FUNCTION_BLOCK FB_Component_Preplate_Rack EXTENDS FB_ComponentBase_SR
VAR_INPUT
    Executing : BOOL;

END_VAR

VAR
    // Inputs

    Button  : FB_Component_Button;
    Closed  : FB_DigitalSensor;
    _InAuto : BOOL;

    // Outputs
    Lock : FB_Component_Indicator;
END_VAR

VAR
    State    : E_RackState;
    R_Button : R_TRIG;

    //Properties
    _Available   : BOOL;
    _LinkBlocked : BOOL;
    _Blocked     : BOOL;
    Linked       : BOOL := TRUE;

    // Alarms
    RackDoorAlarms : ARRAY[1..RACK_DOOR_ALARMS_COUNT] OF FB_TcAlarm;

END_VAR

VAR
    // Internal state variables
    DoorLocked : BOOL := FALSE;
END_VAR

VAR CONSTANT
    RACK_DOOR_ALARMS_COUNT : UDINT := 5;
END_VAR

METHOD Block
VAR_INPUT
    Blocked : BOOL;
END_VAR
_Blocked := Blocked;
END_METHOD

PROPERTY Blocked : BOOL
GET
Blocked := _Blocked;
END_GET
SET
_Blocked := Blocked;
END_SET
END_PROPERTY

//! @summary This method serves as the entry point for all underlying FB logic
METHOD PUBLIC CyclicLogic

//! @description This method should be called cyclically by descendant function blocks by invoking <c>SUPER^.CyclicLogic()</c>.  Alternatively, the contents of this method could be reimplemented entirely in which case a call to this method would not be necessary.
RackLogic();

Button.CyclicLogic();
Closed.CyclicLogic();
Lock.CyclicLogic();

SUPER^.CyclicLogic();
END_METHOD

METHOD Disable
VAR_INPUT
END_VAR
_Available := FALSE;
END_METHOD

PROPERTY PUBLIC InAuto : BOOL
SET
_InAuto := InAuto;
END_SET
END_PROPERTY

//! @summary Basic component initialization logic
METHOD PROTECTED Initialize : BOOL;

//! @description This method is called by <c>CyclicLogic()</c> as required
CreateEvents();

IF SUPER^.Initialize() THEN
    Initialize := TRUE;
END_IF
END_METHOD

METHOD IsAvailable : BOOL
VAR_INPUT
END_VAR
IsAvailable := _Available;
END_METHOD

PROPERTY LinkBlocked : BOOL
GET
LinkBlocked := _LinkBlocked;
END_GET
SET
_LinkBlocked := LinkBlocked;
END_SET
END_PROPERTY

METHOD RackLogic
VAR_INPUT
END_VAR
R_Button(CLK := (Button.Button.Active));

CASE State OF
    E_RackState.Idle:
        Button.LED.TurnOn();
        Lock.TurnOn();
        _Available := TRUE;
        IF R_Button.Q THEN
            State := E_RackState.CheckForBlock;
        END_IF;

    E_RackState.CheckForBlock:
        Button.LED.Flash();
        Lock.TurnOn();
        IF NOT Blocked THEN
            State := E_RackState.CheckForLinked;
        ELSIF R_Button.Q THEN
            State := E_RackState.LockDoor;
        END_IF;

    E_RackState.CheckForLinked:
        Button.LED.Flash();
        IF NOT LinkBlocked THEN
            State := E_RackState.UnlockDoor;
        END_IF;

        IF NOT Linked THEN
            State := E_RackState.UnlockDoor;
        ELSIF R_Button.Q THEN
            State := E_RackState.LockDoor;
        END_IF;

    E_RackState.UnlockDoor:
        Lock.TurnOff();
        Button.LED.Flash();
        _Available := FALSE;
        State      := E_RackState.WaitForOpen;

    E_RackState.WaitForOpen:
        Button.LED.TurnOff();
        IF NOT Closed.Active THEN
            State := E_RackState.WaitForClose;
        END_IF;

    E_RackState.WaitForClose:
        Button.LED.TurnOff();
        IF Closed.Active THEN
            State := E_RackState.LockDoor;
        END_IF;

    E_RackState.LockDoor:
        Lock.TurnOn();
        Button.LED.Flash();
        State := E_RackState.EnableDoor;

    E_RackState.EnableDoor:
        Lock.TurnOn();
        _Available := TRUE;
        State      := E_RackState.Idle;
END_CASE;

IF NOT Executing THEN
    Lock.TurnOff();

END_IF
END_METHOD

END_FUNCTION_BLOCK

(* stored: Version 1.1.0.1
   POU FB_Component_Preplate_Rack: Id {140dffbd-304d-4719-a3a1-216bf5831242}, SpecialFunc None
   Folder I_ComponentBase: Id {e37cfa7c-4528-49df-94c9-fc5af6ad140f}
   Folder I_CyclicFB: Id {5d76e6b8-cac5-44aa-8843-44cf313556b4}
   Folder I_PreplateRack: Id {7ffd7deb-cd66-4056-aeef-03665cc0122b}
   Folder Methods: Id {45e321d8-a239-4eb3-b176-b7f97ea5e0a3}
   Folder Properties: Id {00069080-63ce-4a2e-9cae-f91960191816}
   Method Block: Id {b66f7522-8d97-4258-9335-a16039e4e516}
   Property Blocked: Id {44e86bb0-6511-4bb7-ac3a-2a855d3a0939}
   Get Get: Id {b6bd32aa-f21d-4ad1-8266-efc9edf33d40}
   Set Set: Id {7ff5a8fe-2e0e-41db-af02-88a27a95b2f3}
   Method CyclicLogic: Id {fc886497-fd76-4210-ba29-1a53642dfd16}
   Method Disable: Id {8fb7f0b3-5bce-47f2-9692-287f90893fa5}
   Property InAuto: Id {556d3f89-434a-427f-b06a-2bfcff699a20}
   Set Set: Id {431e2ce9-73a7-4e77-a65d-c6ab2a1d6767}
   Method Initialize: Id {688196a4-7727-47f2-8b56-8dd6ead9680e}
   Method IsAvailable: Id {274b1aa5-92ae-4425-b753-a97cd92313ef}
   Property LinkBlocked: Id {8c3827e8-725b-4c24-ac55-488da1da9138}
   Get Get: Id {85b43550-5b1c-4b82-99f1-67303e77afae}
   Set Set: Id {9236ab0f-421b-41df-8e96-a5403df0bb6e}
   Method RackLogic: Id {3126a4e4-285a-455c-8625-38aebb4fdea2} *)
